// TIA Portal V17 export
// export: Created 2023-12-22T15:05:33.919505Z, ExportSetting WithDefaults, DisplayName Totally Integrated Automation Portal, DisplayVersion V17, DisplayName TIA Portal Openness, DisplayVersion V17, DisplayName TIA Portal Version Control Interface, DisplayVersion V17, DisplayName STEP 7 Professional, DisplayVersion V17, DisplayName STEP 7 Safety, DisplayVersion V17, DisplayName WinCC Advanced, DisplayVersion V17
DATA_BLOCK "ModBus_TCP_DB"   // DB40
VERSION : 0.1
// stored: AutoNumber false, DBAccessibleFromOPCUA true, InstanceOfName ModBus_TCP, InstanceOfType FB
"ModBus_TCP"
   // VAR RETAIN
   //    COM_Control : Struct
   //       Enable { S7_SetPoint := 'True'} : Bool := TRUE;
   //       Start : Bool;
   //       Reset : Bool;
   //       REQ_NDR : Bool;
   //       REQ_DR : Bool;
   //       REQ_Error : Bool;
   //       REQ_Status : Word;
   //       Error_Code : Word;
   //       Status : Int;
   //    END_STRUCT;
   //    CONNECT { S7_SetPoint := 'True'} : TCON_IP_v4;
   // END_VAR
BEGIN
   CONNECT.InterfaceId := 64;
   CONNECT.ID := 1;
   CONNECT.ConnectionType := 11;
   CONNECT.RemoteAddress.ADDR[1] := 192;
   CONNECT.RemoteAddress.ADDR[2] := 168;
   CONNECT.RemoteAddress.ADDR[3] := 0;
   CONNECT.RemoteAddress.ADDR[4] := 10;
   CONNECT.RemotePort := 502;
END_DATA_BLOCK
